INTERFACE ITestEventHandler_UsesEventArgs EXTENDS IEventHandlerBase

METHOD OnThisEvent
VAR_INPUT
    EventArgs : IStreamReader;
END_VAR
END_METHOD

END_INTERFACE

(* stored: Version 1.1.0.1, ProductVersion 3.1.4024.4
   Itf ITestEventHandler_UsesEventArgs: Id {4fc83335-f553-406a-a7a8-50f79ed47892}
   Method OnThisEvent: Id {cb91866d-6680-4475-aa4a-24cf3d438921} *)
